{attribute 'qualified_only'}
VAR_GLOBAL CONSTANT
	cMAXEVENTS : UDINT := 64;
END_VAR

(* stored: Version 1.1.0.1
   GVL GVL_Diagnostic: Id {1679d5f9-795b-070e-13d7-3eb2b1ec2ef8} *)
